(* PLC project io_engine_1d1s, Dassault Systèmes ControlBuild 2024x *)
(* stored: creationDateTime 2023-10-03T11:12:46-01:00 *)

PROGRAM panel
  VAR_OUTPUT
    forwardPB : BOOL := false;
    stopPB : BOOL := false;
  END_VAR

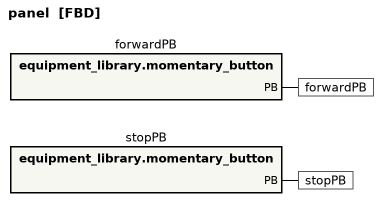
(* FBD diagram, written out as Structured Text *)
forwardPB();
forwardPB := forwardPB.PB;
stopPB();
stopPB := stopPB.PB;
END_PROGRAM

(* Integrated object C/C+OP of a motor with one speed and one direction *)
PROGRAM io_library.io_engine_1d1s
  VAR_INPUT
    autoMode : BOOL := false;
    manualMode : BOOL := false;
  END_VAR
  VAR_INPUT
    autoCmd : BOOL := false;
  END_VAR
  VAR_INPUT
    acknowledgePB : BOOL := false;
  END_VAR
  VAR_OUTPUT
    speedVal : REAL := 0.0;
    speedPercent : REAL := 0.0;
  END_VAR
  VAR_OUTPUT
    generalFault : BOOL := false;
  END_VAR

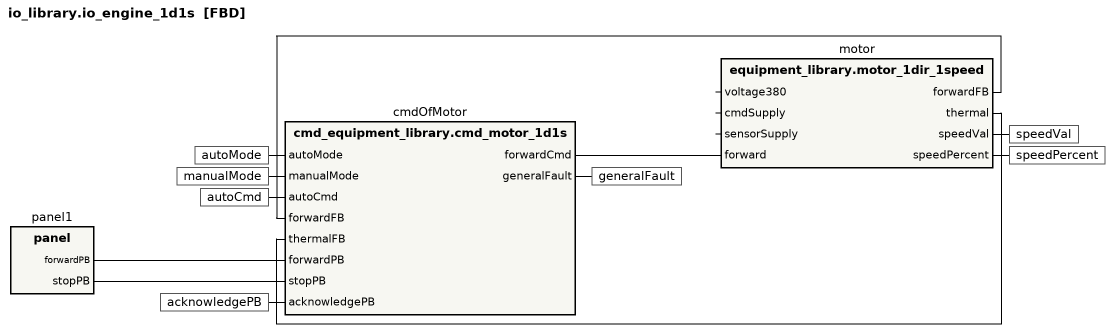
(* FBD diagram, written out as Structured Text *)
motor(forward := cmdOfMotor.forwardCmd);
panel1();
cmdOfMotor(autoMode := autoMode, manualMode := manualMode, autoCmd := autoCmd, forwardFB := motor.forwardFB, thermalFB := motor.thermal, forwardPB := panel1.forwardPB, stopPB := panel1.stopPB, acknowledgePB := acknowledgePB);
generalFault := cmdOfMotor.generalFault;
speedVal := motor.speedVal;
speedPercent := motor.speedPercent;
END_PROGRAM
